VAR_GLOBAL
END_VAR

(* stored: Version 1.1.0.1, ProductVersion 3.1.0.26
   GVL GVLdd: Id {36df5fb0-1b8a-4600-aa9f-ffe0efc22642} *)
